{attribute 'GeneratedUsingTerminal: EL6080-0000-0016'}
{attribute addProperty BoxType "EL6080-0000-0016"}
{attribute addProperty Id "EtcSlaveTerminalBaseStatusAT %I*Status_EF5E6C280InputsEMPTY_STRUCTURE0ControlAT %Q*Control_883019540OutputsEMPTY_STRUCTURE0WcStateAT %I*WcState_9091E0EB2InfoDataAT %I*InfoData_32EB74EA10"}
{attribute addProperty CRC "2629842823"}
{attribute addProperty Size "12"}
TYPE EL6080_9CC03787 EXTENDS EtcSlaveTerminalBase :
STRUCT
	{attribute addProperty Name "Status"}
	Status : Status_EF5E6C28;
	{attribute addProperty Name "Inputs"}
	Inputs : EMPTY_STRUCTURE;
	{attribute addProperty Name "Control"}
	Control : Control_88301954;
	{attribute addProperty Name "Outputs"}
	Outputs : EMPTY_STRUCTURE;
	{attribute addProperty Name "WcState"}
	WcState : WcState_9091E0EB;
	{attribute addProperty Name "InfoData"}
	InfoData : InfoData_32EB74EA;
END_STRUCT
END_TYPE

(* stored: Version 1.2.0.0, ProductVersion 3.1.4024.9
   DUT EL6080_9CC03787: Id {03b34d47-8f80-4a7e-9ee5-66aedb1d6528} *)
